FUNCTION_BLOCK FB_HMI_TIP_A EXTENDS FB_HMI_COMPONENT
VAR_OUTPUT
END_VAR
VAR_IN_OUT
    fbInstance : FB_NOTT_TIP_TILT;
END_VAR
VAR
END_VAR

fbHealthStatus(

    bIsGood := NOT fbInstance.stat.bError,
    bHasWarning := (    fbInstance.stat.bWarning));
                     
fbBusyStatus(

    bIsBusy := FALSE);

M_UpdateStatusColor();

END_FUNCTION_BLOCK

(* stored: Version 1.1.0.1, ProductVersion 3.1.4024.14
   POU FB_HMI_TIP_A: Id {0b2fe298-df1b-4b37-be58-aae3488e7fc9}, SpecialFunc None *)
